TYPE ST_PNOutput_ZPT :
STRUCT
	w_Status					:	WORD;
	w_Warnings					:	WORD;
	w_Faults					:	WORD;
	ui_RatedPower				:	UINT;
	ui_PowerLoad				:	UINT;
	i_TransformerTemperature	:	INT;
END_STRUCT
END_TYPE

(* stored: Version 1.1.0.1, ProductVersion 3.1.4024.12
   DUT ST_PNOutput_ZPT: Id {c765ef42-cb77-41c1-9693-2e3fa15655e5} *)
